Universal Robots URScript: 00B_02_TieXian.script

def P00B_02_TieXian():
  set_standard_analog_input_domain(0, 1)
  set_standard_analog_input_domain(1, 1)
  set_tool_analog_input_domain(0, 1)
  set_tool_analog_input_domain(1, 1)
  set_analog_outputdomain(0, 0)
  set_analog_outputdomain(1, 0)
  set_tool_voltage(0)
  set_input_actions_to_default()
  set_tcp(p[-0.06448999999999999,0.0207,0.28314999999999996,0.0,0.0,1.5902])
  set_payload(8.0)
  set_safety_mode_transition_hardness(1)
  set_gravity([0.0, 0.0, 9.82])
  $ 1 "机器人程序"
  $ 2 "MoveJ"
  $ 3 "路点_1"
  set_tcp(p[-0.06448999999999999,0.0207,0.28314999999999996,0.0,0.0,1.5902])
  movej(get_inverse_kin(p[.827616903570, -.301123339254, .721815651372, -.103069504621, .077854273636, -1.659415960467], qnear=[-0.16091472307314092, -1.8779247442828577, -1.9052231947528284, -1.039285961781637, -1.6081789175616663, 1.6170494556427002]), a=0.6981317007977318, v=0.5235987755982988)
  $ 4 "路点_2"
  set_tcp(p[-0.06448999999999999,0.0207,0.28314999999999996,0.0,0.0,1.5902])
  movej(get_inverse_kin(p[.827602710369, -.301162801291, 1.000581485497, -.103027200423, .077828406675, -1.659426590982], qnear=[-0.16183835664858037, -1.6981428305255335, -1.5959895292865198, -1.5283563772784632, -1.6082266012774866, 1.614162802696228]), a=0.6981317007977318, v=0.5235987755982988)
end
